Fanuc KAREL source: port_GOUT.kl

PROGRAM TP
%NOLOCKGROUP
VAR
 x: INTEGER
BEGIN
 x = GOUT[3]
END TP
